{region '#Template'}
	{attribute 'Version' := '1.0.0.0'}
	{attribute 'Tags' := '"LCID": "1031", "Text": "Universal, Motor, Aggregate"'}
	{attribute 'Tags' := '"LCID": "1033", "Text": "Universal, Motor, Aggregate"'}
	{attribute 'Description' := '"LCID": "1031", "Text": "Motor modulierend mit Regler erweitert"'}
	{attribute 'Description' := '"LCID": "1033", "Text": "Motor modulating with controller extended"'}
{endregion}		 
FUNCTION_BLOCK FB_BA_MotCtlExt EXTENDS FB_BA_AggregateMB
VAR_INPUT
	fIn				: REAL;
END_VAR
VAR_INPUT CONSTANT PERSISTENT
	{attribute 'parameterCategory' := 'Behaviour'}
	fMinModulation : REAL := 20;
	{attribute 'parameterCategory' := 'Behaviour'}
	fMaxModulation : REAL := 100;
END_VAR
VAR_OUTPUT
	bCmd			: BOOL;
	fMdlt			: REAL;
END_VAR
VAR
	eValSfty		: REFERENCE TO E_BA_MdltCmd	REF= nValSfty;
	eValCrit		: REFERENCE TO E_BA_MdltCmd	REF= nValCrit;
	eValPgm			: REFERENCE TO E_BA_MdltCmd	REF= nValPgm;
	eActiveVal		: REFERENCE TO E_BA_MdltCmd	REF= nActiveVal;
END_VAR
VAR_INPUT CONSTANT
	Dst				: FB_BA_BI_IO;
	ThOvrld			: FB_BA_BI_IO;							
	MntnSwi			: FB_BA_BI_IO;							
	Cmd				: FB_BA_BO_IO;								 
	Mdlt			: FB_BA_AO_IO;							
	Sp				: FB_BA_AV_Op;		 
	Ctrl			: FB_BA_Loop;									
END_VAR
VAR
	MuxCmd			: FB_BA_MMUX_B04;
	MuxMdlt			: FB_BA_MMUX_R04;
	fMax			: REAL;
	fMin			: REAL;		
END_VAR

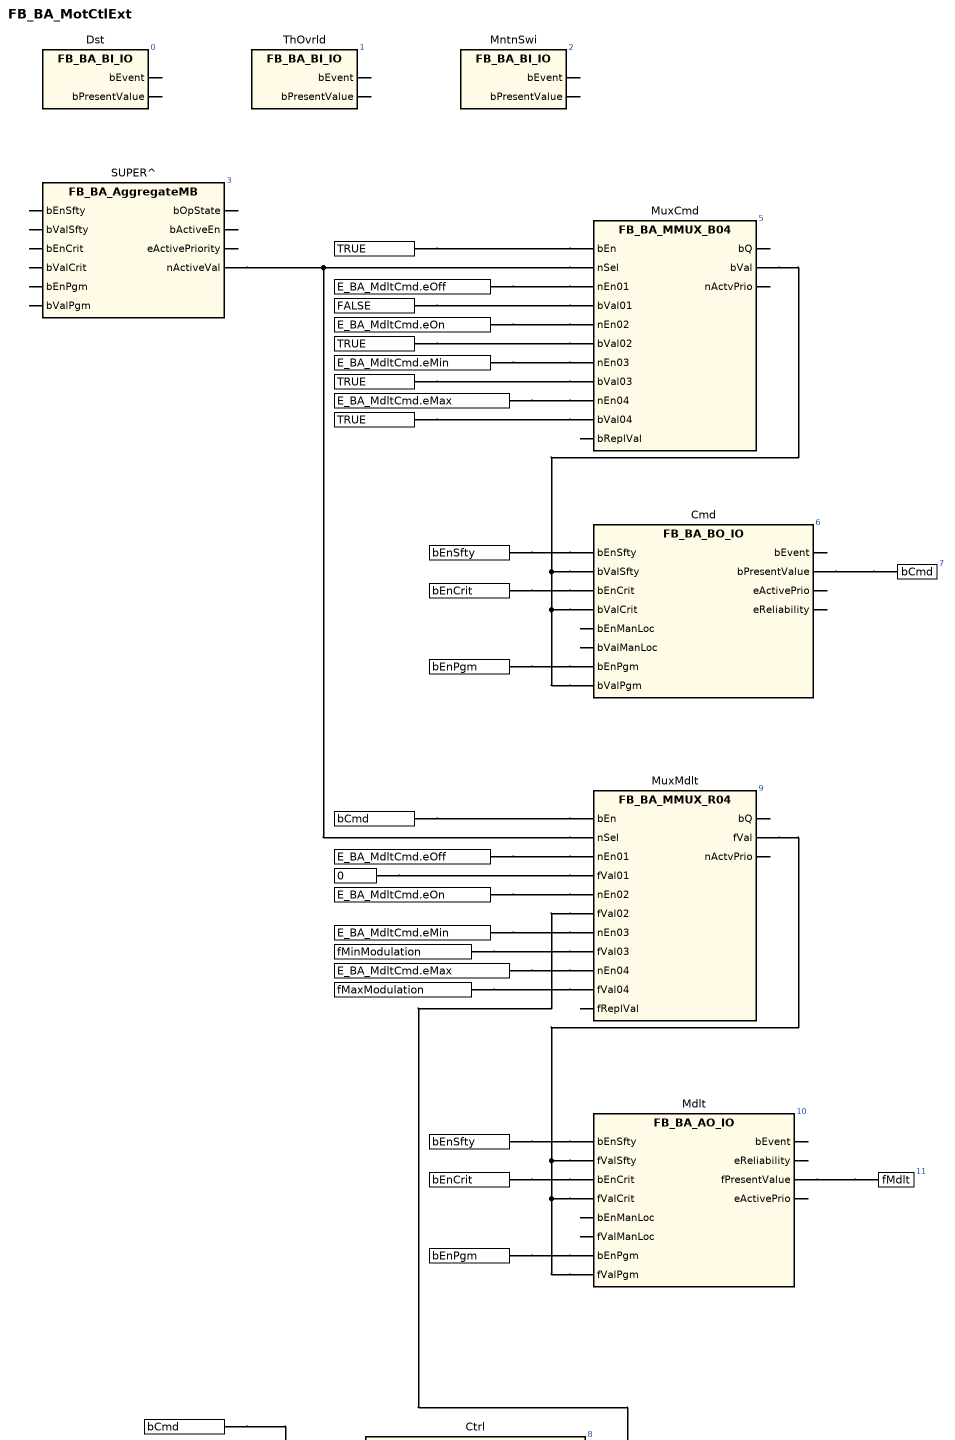
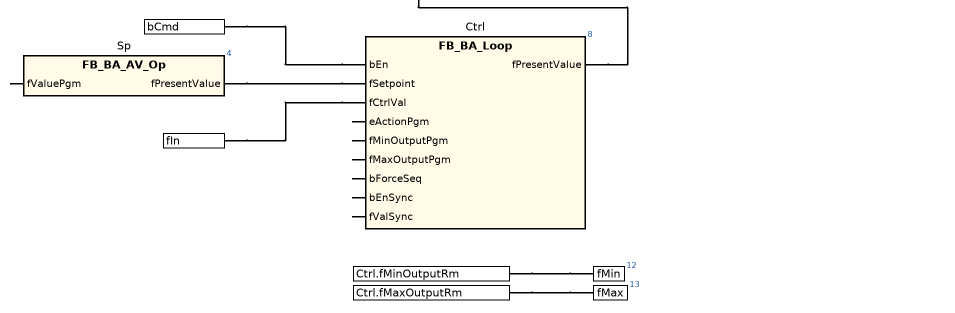
Dst(); // FB_BA_BI_IO
ThOvrld(); // FB_BA_BI_IO
MntnSwi(); // FB_BA_BI_IO
SUPER^(); // FB_BA_AggregateMB
Sp(); // FB_BA_AV_Op
MuxCmd(
    bEn := TRUE,
    nSel := SUPER^.nActiveVal,
    nEn01 := E_BA_MdltCmd.eOff,
    bVal01 := FALSE,
    nEn02 := E_BA_MdltCmd.eOn,
    bVal02 := TRUE,
    nEn03 := E_BA_MdltCmd.eMin,
    bVal03 := TRUE,
    nEn04 := E_BA_MdltCmd.eMax,
    bVal04 := TRUE); // FB_BA_MMUX_B04
Cmd(
    bEnSfty := bEnSfty,
    bValSfty := MuxCmd.bVal,
    bEnCrit := bEnCrit,
    bValCrit := MuxCmd.bVal,
    bEnPgm := bEnPgm,
    bValPgm := MuxCmd.bVal); // FB_BA_BO_IO
bCmd := Cmd.bPresentValue;
Ctrl(bEn := bCmd, fSetpoint := Sp.fPresentValue, fCtrlVal := fIn); // FB_BA_Loop
MuxMdlt(
    bEn := bCmd,
    nSel := SUPER^.nActiveVal,
    nEn01 := E_BA_MdltCmd.eOff,
    fVal01 := 0,
    nEn02 := E_BA_MdltCmd.eOn,
    fVal02 := Ctrl.fPresentValue,
    nEn03 := E_BA_MdltCmd.eMin,
    fVal03 := fMinModulation,
    nEn04 := E_BA_MdltCmd.eMax,
    fVal04 := fMaxModulation); // FB_BA_MMUX_R04
Mdlt(
    bEnSfty := bEnSfty,
    fValSfty := MuxMdlt.fVal,
    bEnCrit := bEnCrit,
    fValCrit := MuxMdlt.fVal,
    bEnPgm := bEnPgm,
    fValPgm := MuxMdlt.fVal); // FB_BA_AO_IO
fMdlt := Mdlt.fPresentValue;
fMin := Ctrl.fMinOutputRm;
fMax := Ctrl.fMaxOutputRm;

METHOD FB_init : BOOL
VAR_INPUT
	bInitRetains : BOOL; // if TRUE, the retain variables are initialized (warm start / cold start)
	bInCopyCode : BOOL;  // if TRUE, the instance afterwards gets moved into the copy code (online change)
END_VAR
Dst.iParent							:= THIS^;
Dst.iLabel							:= LblUniFieldDevice.Motor_Dst;	
Dst.sObjectName						:= '{Idx=01}';	
Dst.sDeviceType						:= '';
Dst.bEnOutOfService					:= FALSE;
Dst.ePolarity						:= E_BA_Polarity.eReverse;
Dst.sActiveText 					:= txtEvent_Triggered;
Dst.sInactiveText 					:= txtEvent_Normal;
Dst.nStateChangeCount				:= 0;
Dst.nActiveTimeElapsed				:= 0;
Dst.nEventClassID					:= EventClasses.AlarmTechnicalExtended;
Dst.stTimeDelay.nToNormal			:= BA2_Param.nDefTimeDelay_ToNormal;
Dst.stTimeDelay.nToAbnormal			:= BA2_Param.nDefTimeDelay_ToAbnormal;
Dst.bAlarmValue						:= TRUE;
Dst.bAcknowledgeRm					:= FALSE;	
Dst.aEventTransitionText[1]			:= txtEvent_Triggered;
Dst.aEventTransitionText[2]			:= txtEvent_Error;
Dst.aEventTransitionText[3]			:= txtEvent_Normal;
Dst.bEventDetectionEnable			:= TRUE;
Dst.eEnPlantLock					:= E_BA_LockPriority.eLocalMedium;

ThOvrld.iParent						:= THIS^;
ThOvrld.iLabel						:= LblUniFieldDevice.Motor_Dst;	
ThOvrld.sObjectName					:= '{Idx=02}';	
ThOvrld.sDeviceType					:= '';
ThOvrld.bEnOutOfService				:= FALSE;
ThOvrld.ePolarity					:= E_BA_Polarity.eReverse;
ThOvrld.sActiveText 				:= txtEvent_Triggered;
ThOvrld.sInactiveText 				:= txtEvent_Normal;
ThOvrld.nStateChangeCount			:= 0;
ThOvrld.nActiveTimeElapsed			:= 0;
ThOvrld.nEventClassID				:= EventClasses.AlarmTechnicalExtended;
ThOvrld.stTimeDelay.nToNormal		:= BA2_Param.nDefTimeDelay_ToNormal;
ThOvrld.stTimeDelay.nToAbnormal		:= BA2_Param.nDefTimeDelay_ToAbnormal;
ThOvrld.bAlarmValue					:= TRUE;
ThOvrld.bAcknowledgeRm				:= FALSE;	
ThOvrld.aEventTransitionText[1]		:= txtEvent_Triggered;
ThOvrld.aEventTransitionText[2]		:= txtEvent_Error;
ThOvrld.aEventTransitionText[3]		:= txtEvent_Normal;
ThOvrld.bEventDetectionEnable		:= TRUE;
ThOvrld.eEnPlantLock				:= E_BA_LockPriority.eLocalMedium;	

MntnSwi.iParent						:= THIS^;
MntnSwi.iLabel						:= LblUniFieldDevice.Motor_MntnSwi;	
MntnSwi.sObjectName					:= '{Idx=01}';
MntnSwi.sDeviceType					:= '';
MntnSwi.bEnOutOfService				:= FALSE;	
MntnSwi.ePolarity					:= E_BA_Polarity.eReverse;
MntnSwi.sActiveText 				:= txtEvent_Maintenace;
MntnSwi.sInactiveText 				:= txtEvent_Normal;
MntnSwi.nStateChangeCount			:= 0;
MntnSwi.nActiveTimeElapsed			:= 0;
MntnSwi.nEventClassID				:= EventClasses.MaintenanceSimple;
MntnSwi.stTimeDelay.nToNormal		:= BA2_Param.nDefTimeDelay_ToNormal;
MntnSwi.stTimeDelay.nToAbnormal		:= BA2_Param.nDefTimeDelay_ToAbnormal;
MntnSwi.bAlarmValue					:= TRUE;
MntnSwi.bAcknowledgeRm				:= FALSE;	
MntnSwi.aEventTransitionText[1]		:= txtEvent_Disturb;
MntnSwi.aEventTransitionText[2]		:= txtEvent_None;
MntnSwi.aEventTransitionText[3]		:= txtEvent_Normal;
MntnSwi.bEventDetectionEnable		:= TRUE;
MntnSwi.eEnPlantLock				:= E_BA_LockPriority.eLocalMedium;

Cmd.iParent							:= THIS^;
Cmd.iLabel							:= LblUniFieldDevice.Motor_Cmd;			
Cmd.sObjectName						:= '{Idx=01}';	
Cmd.sDeviceType						:= '';
Cmd.bEnOutOfService					:= FALSE;
Cmd.ePolarity						:= E_BA_Polarity.eNormal;
Cmd.eFeedbackPolarity				:= E_BA_Polarity.eNormal;
Cmd.eOverriddenPolarity				:= E_BA_Polarity.eReverse;
Cmd.sActiveText 					:= txtEvent_On;
Cmd.sInactiveText 					:= txtEvent_Off;
Cmd.nStateChangeCount				:= 0;
Cmd.nActiveTimeElapsed				:= 0;
Cmd.nMinimumOnTime					:= 0;
Cmd.nMinimumOffTime					:= 0;
Cmd.bEnManualRm						:= FALSE;	//	Priority  8	
Cmd.bValManualRm					:= FALSE;	//	Priority  8
Cmd.bDefaultValue					:= FALSE;
Cmd.nEventClassID					:= EventClasses.DisturbanceExtended;
Cmd.stTimeDelay.nToNormal			:= BA2_Param.nDefTimeDelay_ToNormal;
Cmd.stTimeDelay.nToAbnormal			:= BA2_Param.nDefTimeDelay_ToAbnormal;
Cmd.bAcknowledgeRm					:= FALSE;		
Cmd.aEventTransitionText[1]			:= txtEvent_Disturb;
Cmd.aEventTransitionText[2]			:= txtEvent_None;
Cmd.aEventTransitionText[3]			:= txtEvent_Normal;
Cmd.bEventDetectionEnable			:= FALSE;
Cmd.eEnPlantLock					:= E_BA_LockPriority.eNoLock;

Mdlt.iParent						:= THIS^;
Mdlt.iLabel							:= LblUniFieldDevice.Motor_Mdlt;	
Mdlt.sObjectName					:= '{Idx=01}';
Mdlt.sDeviceType					:= '';
Mdlt.bEnOutOfService				:= FALSE;
Mdlt.eOverriddenPolarity			:= E_BA_Polarity.eNormal;
Mdlt.eUnit							:= E_BA_Unit.eOther_Percent;
Mdlt.fResolution 					:= 0.003051851;
Mdlt.fScaleOffset 					:= 0;
Mdlt.fCOVIncrement					:= BA2_Param.fDefCOVIncrement;
Mdlt.bEnManualRm					:= FALSE;	//	Priority  8	
Mdlt.fValManualRm					:= 0.0;		//	Priority  8
Mdlt.fDefaultValue					:= 0.0;	
Mdlt.nEventClassID					:= EventClasses.NotificationSimple;
Mdlt.stTimeDelay.nToNormal			:= BA2_Param.nDefTimeDelay_ToNormal;
Mdlt.stTimeDelay.nToAbnormal		:= BA2_Param.nDefTimeDelay_ToAbnormal;
Mdlt.stHighLimit.bEnable			:= FALSE;
Mdlt.stHighLimit.fValue				:= 0.0;		
Mdlt.stLowLimit.bEnable				:= FALSE;
Mdlt.stLowLimit.fValue				:= 0.0;
Mdlt.fLimitDeadband 				:= BA2_Param.fDefLimitDeadband;
Mdlt.bAcknowledgeRm					:= FALSE;	
Mdlt.aEventTransitionText[1]		:= txtEvent_Disturb;
Mdlt.aEventTransitionText[2]		:= txtEvent_None;
Mdlt.aEventTransitionText[3]		:= txtEvent_Normal;
Mdlt.bEventDetectionEnable			:= FALSE;
Mdlt.eEnPlantLock					:= E_BA_LockPriority.eNoLock;

Sp.iParent							:= THIS^;
Sp.iLabel							:= LblUniFieldDevice.Motor_Sp;		
Sp.sObjectName						:= '{Idx=01}';								 	 
Sp.eUnit 							:= E_BA_Unit.ePressure_Pascals;								 
Sp.fValueRm							:= 250;
Sp.fCOVIncrement					:= BA2_Param.fDefCOVIncrement;

Ctrl.iParent						:= THIS^;
Ctrl.iLabel							:= LblUniFieldDevice.Motor_Ctrl; 
Ctrl.sObjectName					:= '{Idx=01}';
Ctrl.eOpMode						:= BA2_Param.nLoop_DefOpMode;								 	 										 
Ctrl.eOutputUnit					:= E_BA_Unit.eOther_Percent;
Ctrl.eActionRm						:= E_BA_Action.eReverse;
Ctrl.fProportionalConstant			:= 0.01;
Ctrl.fIntegralConstant				:= 60;
Ctrl.fDerivativeConstant			:= 0;
Ctrl.fMaxOutputRm 					:= 100;
Ctrl.fMinOutputRm					:= 20;
Ctrl.fCOVIncrement					:= 0;
Ctrl.nDampConstant					:= 0;
Ctrl.fNeutralZone					:= 0;
END_METHOD

END_FUNCTION_BLOCK

(* stored: Version 1.1.0.1, ProductVersion 3.1.4024.9
   POU FB_BA_MotCtlExt: Id {cb1c2702-93d0-41c1-a114-ec0b657e25be}, SpecialFunc None
   Method FB_init: Id {4a5ad6bc-ecfd-46a4-8c6d-838a8355bf7b} *)
